FUNCTION_BLOCK Product2
  (* Version 1.0, 2008-11-05, Goran Cengic, Chalmers *)
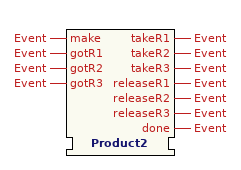
  EVENT_INPUT
    make;
    gotR1;
    gotR2;
    gotR3;
  END_EVENT
  EVENT_OUTPUT
    takeR1;
    takeR2;
    takeR3;
    releaseR1;
    releaseR2;
    releaseR3;
    done;
  END_EVENT
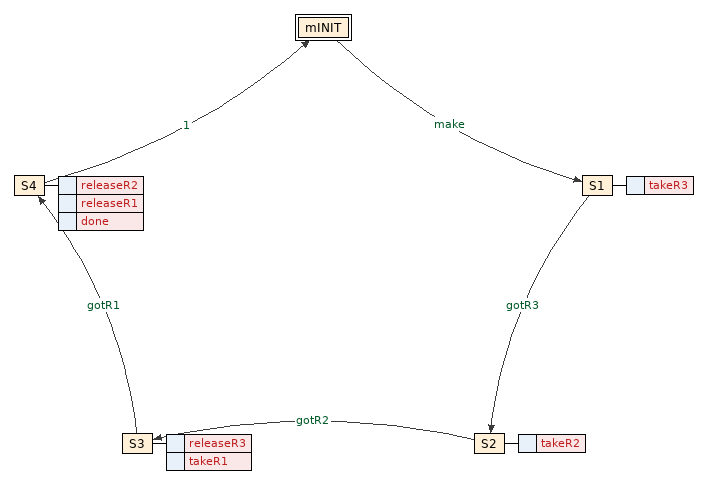
  EC_STATES
    mINIT;
    S1 : -> takeR3;
    S2 : -> takeR2;
    S3 : -> releaseR3, -> takeR1;
    S4 : -> releaseR2, -> releaseR1, -> done;
  END_STATES
  EC_TRANSITIONS
    mINIT TO S1 := make;
    S1 TO S2 := gotR3;
    S2 TO S3 := gotR2;
    S3 TO S4 := gotR1;
    S4 TO mINIT := 1;
  END_TRANSITIONS
END_FUNCTION_BLOCK
